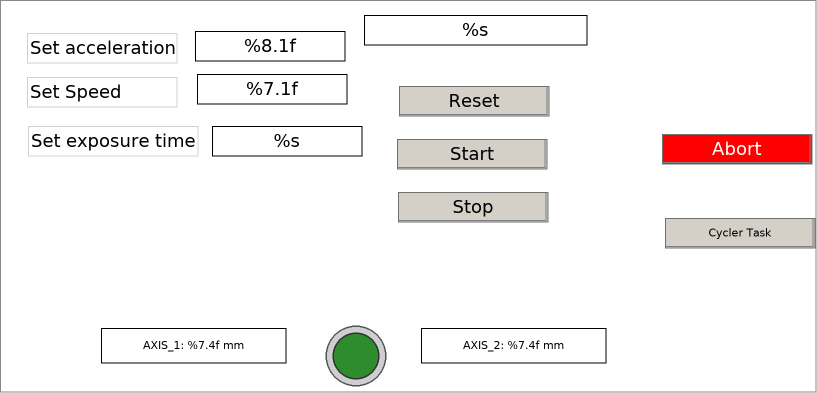
VISUALIZATION CyclerGUI  // 817x393
    Button (399,86 150x30), "Reset", input disabled if: MAIN.cycler.state <> ShutterState.STOPPED
        OnMouseUp: execute { MAIN.reset := TRUE; }
    Button (662,134 150x30), "Abort"
        OnMouseUp: execute { MAIN.abort := TRUE; }
    Button (397,139 150x30), "Start", input disabled if: MAIN.cycler.state <> ShutterState.STOPPED
        OnMouseUp: execute { MAIN.start := TRUE; }
    Button (398,192 150x30), "Stop", input disabled if: MAIN.cycler.state < ShutterState.OPENING
        OnMouseUp: execute { MAIN.stop := TRUE; }
    Rectangle (364,15 223x30), "%s", text variable: MAIN.cycler.state
    Textfield (27,33 150x30), "Set acceleration", input disabled if: MAIN.cycler.state <> ShutterState.STOPPED
        OnMouseUp: write MAIN.acceleration via Default, min 0, max 20000, format %8.1f
    Textfield (27,77 150x30), "Set Speed", input disabled if: MAIN.cycler.state <> ShutterState.STOPPED
        OnMouseUp: write MAIN.speed via Default, min 0, max 2000, format %7.1f
    Textfield (28,126 170x30), "Set exposure time", input disabled if: MAIN.cycler.state <> ShutterState.STOPPED
        OnMouseDown: write MAIN.exposure via Default, min T#0s, max T#30s
    Rectangle (195,31 150x30), "%8.1f", text variable: MAIN.acceleration
    Rectangle (197,74 150x30), "%7.1f", text variable: MAIN.speed
    Rectangle (212,126 150x30), "%s", text variable: MAIN.exposure
    Lamp1 (321,321 70x70), variable: GVL.brakeRelays = 3, style: Lamp-Lamp1-Green
    Rectangle (101,328 185x35), "AXIS_1: %7.4f mm", text variable: MAIN.physicalAxes[0].NcToPlc.ActPos
    Rectangle (421,328 185x35), "AXIS_2: %7.4f mm", text variable: MAIN.physicalAxes[1].NcToPlc.ActPos
    Button (665,218 150x30), "Cycler Task", input disabled if: GVL.task=1;
        OnMouseUp: execute { GVL.task:=1; }
END_VISUALIZATION

(* stored: Version 1.1.0.1, ProductVersion 3.1.4020.12
   Visu CyclerGUI: Id {e5c2829f-ff65-484d-a726-9a2e79865c92} *)
